// Mitsubishi GX Works2 project: Feilhåndtering-demo_6   PLC: FX3U/FX3UC

// global labels: Global1
VAR_GLOBAL
  Tank_level AT D300 : INT;
  Tank_high AT Y024 : BOOL;
  Tank_low AT Y002 : BOOL;
  Tank_high_high AT Y003 : BOOL;
  Tank_low_low AT Y004 : BOOL;
  Tank_criticalHigh AT Y006 : BOOL;
  Tank_criticalLow AT Y007 : BOOL;
  Pump AT Y012 : BOOL;
  Set_point AT D302 : INT;
  ErrorSignal AT D304 : WORD;
  Communication_trouble AT X001 : BOOL;
  Communication_troubleRST AT Y001 : BOOL;
  Communication_troubleRSTCommand AT X021 : BOOL;
  Communication_rstFlag AT M1 : BOOL;
  Profibus_code AT D305 : INT;
  Tank_normalHigh AT Y014 : BOOL;
  Tank_normalLow AT Y015 : BOOL;
  Acknowledge_normalHigh AT Y010 : BOOL;
  Acknowledge_normalLow AT Y026 : BOOL;
  Acknowledge_criticalHigh AT Y011 : BOOL;
  Acknowledge_criticalLow AT Y027 : BOOL;
  Process_memory AT M501 : BOOL;
  Process AT Y021 : BOOL;
  Power_failure AT Y022 : BOOL;
  Acknowledge_powerFailure AT Y023 : BOOL;
  Normal_ErrorSignal AT Y030 : BOOL;
  Critical_ErrorSignal AT Y031 : BOOL;
  Normal_ErrorCheck AT M550 : ARRAY [0..2] OF BOOL;
  Critical_ErrorCheck AT M553 : ARRAY [0..2] OF BOOL;
END_VAR

// task Task_01 (event TRUE, interval 0, priority 31): Fault_handling_Signal_Error

PROGRAM Fault_handling_Water_Tank
VAR
  Fault_normal : BOOL;
END_VAR
(* structured ladder/FBD written out as ST: instructions are called as NAME(EN, inputs, outputs); _pN, _eN, _tN stand for wires *)
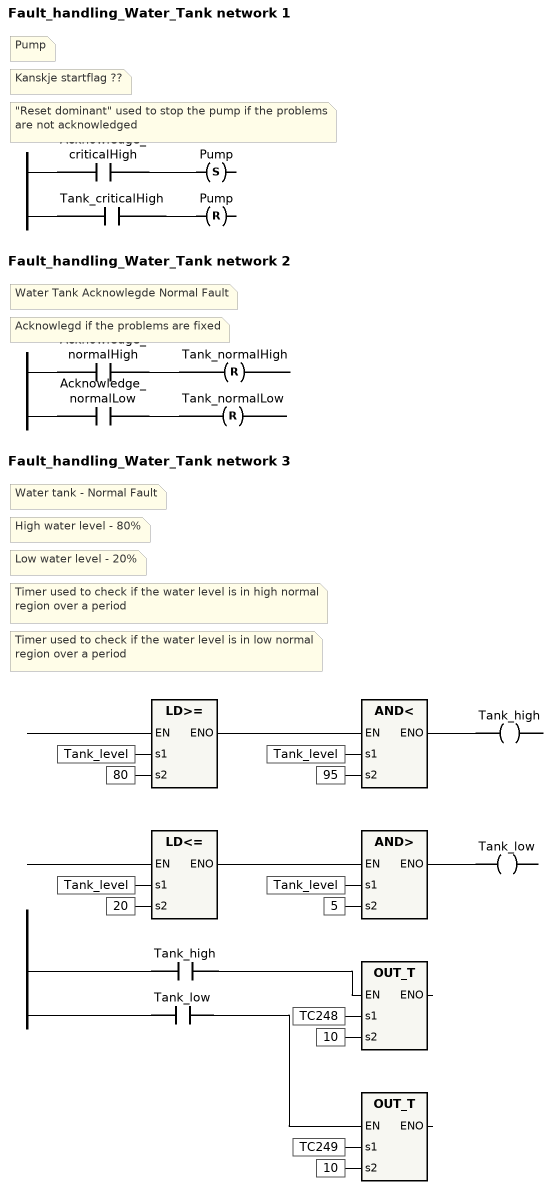
(* network 1 *)
(* Pump *)
(* Kanskje startflag ?? *)
(* "Reset dominant" used to stop the pump if the problems are not acknowledged *)
SET(Acknowledge_criticalHigh, Pump);
RST(Tank_criticalHigh, Pump);
(* network 2 *)
(* Water Tank Acknowlegde Normal Fault *)
(* Acknowlegd if the problems are fixed *)
RST(Acknowledge_normalHigh, Tank_normalHigh);
RST(Acknowledge_normalLow, Tank_normalLow);
(* network 3 *)
(* Water tank - Normal Fault *)
(* High water level - 80% *)
(* Low water level - 20% *)
(* Timer used to check if the water level is in high normal region over a period *)
(* Timer used to check if the water level is in low normal region over a period *)
_e1 := LD>=(TRUE, Tank_level, 80);
_e2 := AND<(_e1, Tank_level, 95);
Tank_high := _e2;
_e3 := LD<=(TRUE, Tank_level, 20);
_e4 := AND>(_e3, Tank_level, 5);
Tank_low := _e4;
OUT_T(Tank_high, TC248, 10);
OUT_T(Tank_low, TC249, 10);
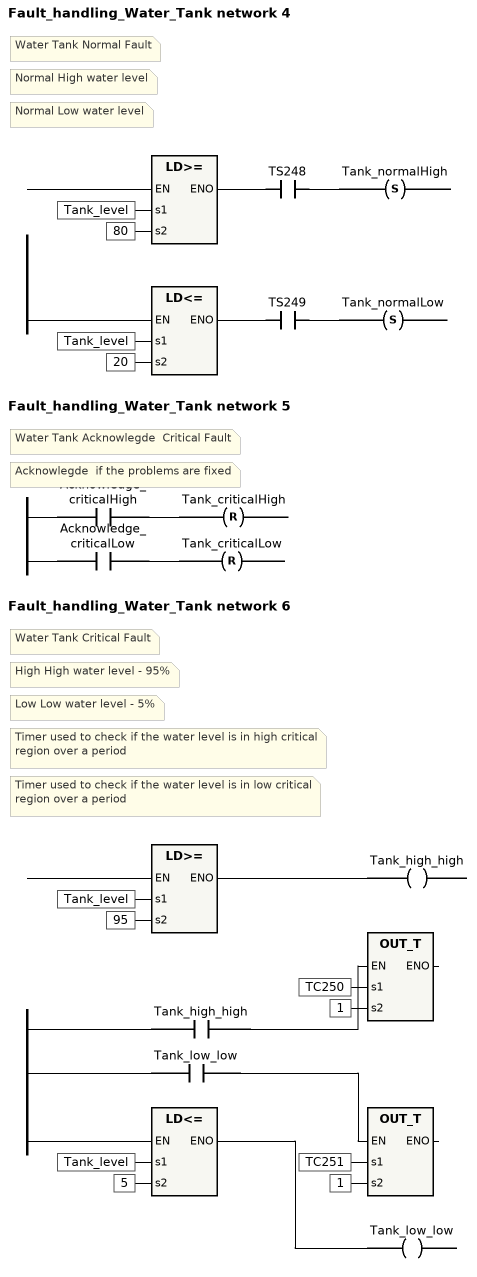
(* network 4 *)
(* Water Tank Normal Fault *)
(* Normal High water level *)
(* Normal Low water level *)
_e1 := LD>=(TRUE, Tank_level, 80);
SET(_e1 AND TS248, Tank_normalHigh);
_e2 := LD<=(TRUE, Tank_level, 20);
SET(_e2 AND TS249, Tank_normalLow);
(* network 5 *)
(* Water Tank Acknowlegde  Critical Fault *)
(* Acknowlegde  if the problems are fixed *)
RST(Acknowledge_criticalHigh, Tank_criticalHigh);
RST(Acknowledge_criticalLow, Tank_criticalLow);
(* network 6 *)
(* Water Tank Critical Fault *)
(* High High water level - 95% *)
(* Low Low water level - 5% *)
(* Timer used to check if the water level is in high critical region over a period *)
(* Timer used to check if the water level is in low critical region over a period *)
_e1 := LD>=(TRUE, Tank_level, 95);
Tank_high_high := _e1;
_e2 := LD<=(TRUE, Tank_level, 5);
Tank_low_low := _e2;
OUT_T(Tank_high_high, TC250, 1);
OUT_T(Tank_low_low, TC251, 1);
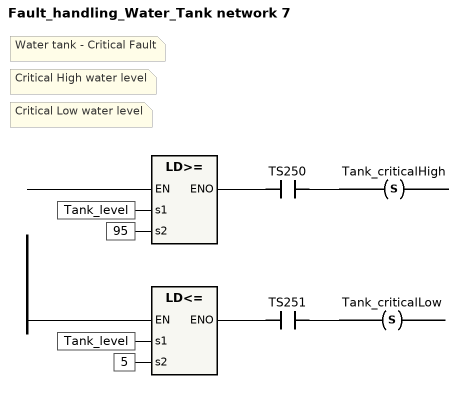
(* network 7 *)
(* Water tank - Critical Fault *)
(* Critical High water level *)
(* Critical Low water level *)
_e1 := LD>=(TRUE, Tank_level, 95);
SET(_e1 AND TS250, Tank_criticalHigh);
_e2 := LD<=(TRUE, Tank_level, 5);
SET(_e2 AND TS251, Tank_criticalLow);
END_PROGRAM

PROGRAM Fault_handling_Signal_Error
VAR
  Normal_Error : BOOL;
  Critical_Error : BOOL;
END_VAR
(* structured ladder/FBD written out as ST: instructions are called as NAME(EN, inputs, outputs); _pN, _eN, _tN stand for wires *)
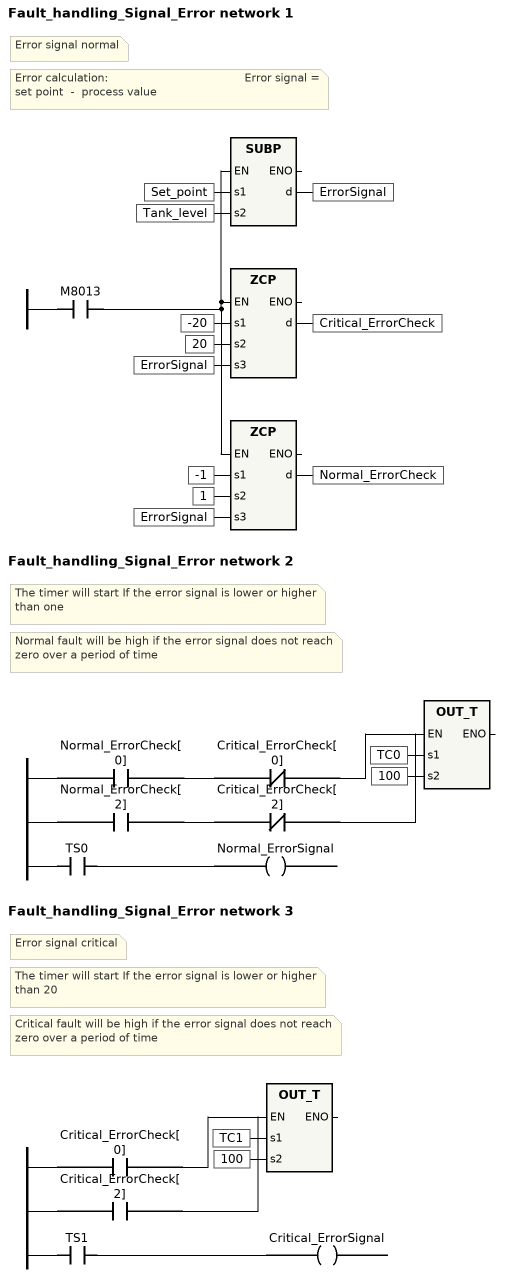
(* network 1 *)
(* Error signal normal *)
(* Error calculation:                                       Error signal = set point  -  process value *)
SUBP(M8013, Set_point, Tank_level, ErrorSignal);
ZCP(M8013, -20, 20, ErrorSignal, Critical_ErrorCheck);
ZCP(M8013, -1, 1, ErrorSignal, Normal_ErrorCheck);
(* network 2 *)
(* The timer will start If the error signal is lower or higher than one *)
(* Normal fault will be high if the error signal does not reach zero over a period of time *)
OUT_T((Normal_ErrorCheck[0] AND NOT Critical_ErrorCheck[0]) OR (Normal_ErrorCheck[2] AND NOT Critical_ErrorCheck[2]), TC0, 100);
Normal_ErrorSignal := TS0;
(* network 3 *)
(* Error signal critical *)
(* The timer will start If the error signal is lower or higher than 20 *)
(* Critical fault will be high if the error signal does not reach zero over a period of time *)
OUT_T(Critical_ErrorCheck[0] OR Critical_ErrorCheck[2], TC1, 100);
Critical_ErrorSignal := TS1;
END_PROGRAM

PROGRAM Fault_handling_Profibus
(* structured ladder/FBD written out as ST: instructions are called as NAME(EN, inputs, outputs); _pN, _eN, _tN stand for wires *)
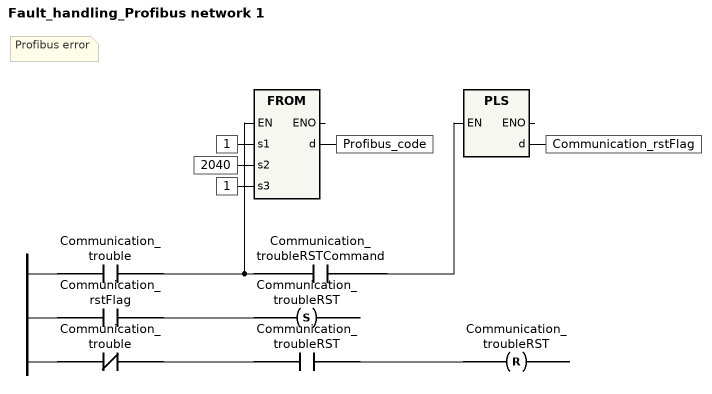
(* network 1 *)
(* Profibus error *)
FROM(Communication_trouble, 1, 2040, 1, Profibus_code);
PLS(Communication_trouble AND Communication_troubleRSTCommand, Communication_rstFlag);
SET(Communication_rstFlag, Communication_troubleRST);
RST(NOT Communication_trouble AND Communication_troubleRST, Communication_troubleRST);
END_PROGRAM

PROGRAM Power_failure
(* structured ladder/FBD written out as ST: instructions are called as NAME(EN, inputs, outputs); _pN, _eN, _tN stand for wires *)
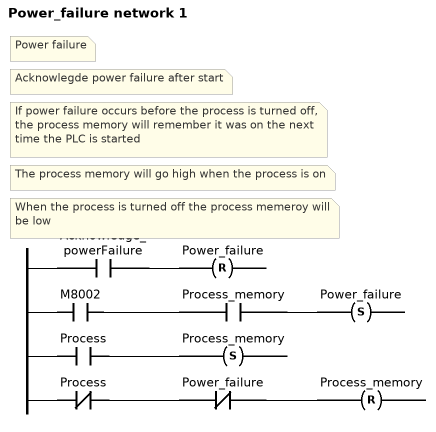
(* network 1 *)
(* Power failure *)
(* Acknowlegde power failure after start *)
(* If power failure occurs before the process is turned off, the process memory will remember it was on the next time the PLC is started *)
(* The process memory will go high when the process is on *)
(* When the process is turned off the process memeroy will be low *)
RST(Acknowledge_powerFailure, Power_failure);
SET(M8002 AND Process_memory, Power_failure);
SET(Process, Process_memory);
RST(NOT Process AND NOT Power_failure, Process_memory);
END_PROGRAM
